{attribute addProperty BoxType "EK1100-0000-0018"}
{attribute addProperty Id "Beckhoff_EQ1xxxEK1122Beckhoff_EQ1xxxEK1122_544C30AD62478"}
{attribute addProperty CRC "2022488474"}
{attribute addProperty SizeInBites "624"}
{attribute addProperty SizeInBytes "78"}
TYPE Beckhoff_EQ1xxx_788CB99A EXTENDS EK1100_179A0949 :
STRUCT
	{attribute addProperty Name "Beckhoff_EQ1xxxEK1122"}
	Beckhoff_EQ1xxxEK1122 : Beckhoff_EQ1xxxEK1122_544C30AD;
END_STRUCT
END_TYPE

(* stored: Version 1.2.0.0, ProductVersion 3.1.4024.9
   DUT Beckhoff_EQ1xxx_788CB99A: Id {35743fd7-a3ef-4897-b73d-5421a5ac38ec} *)
